(* IEC 61131-3 sources: SIMERLIFT/LOGICAD/SIMERLIFT/src_FBD/BCU/CAN/BCU, 3 files *)

(* ---- BCU_Battery_Status.iecfbd ---- *)
FUNCTION_BLOCK BCU_Battery_Status
  {
    SoC {index := 2};
    SoH {index := 3};
    Duty_Cycle {index := 4};
    Remain_Energy {index := 6};
    CAN_CH {index := 0};
    CAN_ID {index := 1};
    CAN_Error {index := 6};
    Available_Energy {index := 5};
    width := 500;
    height := 138;
    bgColor := "cadetblue";
  }

  VAR
    CANSEND4 : CANSEND;
  END_VAR
  VAR_INPUT
    SoC : USINT := 0;
    SoH : USINT := 0;
    Duty_Cycle : UINT := 0;
    Remain_Energy : REAL := 0;
    CAN_ID : UDINT := 0;
    CAN_CH : UDINT := 0;
    Available_Energy : REAL;
  END_VAR
  VAR_OUTPUT
    CAN_Error : BOOL := 0;
  END_VAR

  (*

    // Network 1:
    TO_LWORD(IN := SoC, TO_LWORD => @C(24).TO_LWORD);
    WBIT(start := 0, len := 8, INbit := @C(24).TO_LWORD, OUTbit => @C(2).OUTbit);
    TO_LWORD(IN := SoH, TO_LWORD => @C(31).TO_LWORD);
    WBIT(start := 8, len := 8, INbit := @C(31).TO_LWORD, OUTbit => @C(6).OUTbit);
    NE(IN1 := CAN_ID, IN2 := 0, NE => @C(64).NE);
    TO_LWORD(IN := Duty_Cycle, TO_LWORD => @C(32).TO_LWORD);
    WBIT(start := 16, len := 16, INbit := @C(32).TO_LWORD, OUTbit => @C(10).OUTbit);
    WFLT(start := 32, len := 16, prm := Remain_Energy, ofs := 0, res := 0.01, OUTbit => @C(14).OUTbit);
    WFLT(start := 48, len := 16, prm := Available_Energy, ofs := 0, res := 0.01, OUTbit => @C(15).OUTbit);
    OR(IN1 := @C(2).OUTbit, IN2 := @C(6).OUTbit, IN3 := @C(10).OUTbit, IN4 := @C(14).OUTbit, IN5 := @C(15).OUTbit, OR => @C(12).OR);
    CANSEND4(CH := CAN_CH, ID := CAN_ID, FMT := CAN_FORMAT#EXTENDED, DATA := @C(12).OR, DLC := 8, PER := T#100ms, ENB := @C(64).NE);
    NE(IN1 := CANSEND4.RC, IN2 := 0, NE => CAN_Error);

  *)

  @C(12) : @F(OR), @R(970.0, 60.0, 40.0, 108.0), LWORD, @I(@N(IN1), @L(9.5)), @I(@N(IN2), @L(29.5)), @I(@N(IN3), @L(49.5)), @I(@N(IN4), @L(69.5)), @I(@N(IN5), @L(89.5)), @O(@N(OR), @R(9.5));
  @VF(18) : @E(T#100ms), @R(1160.0, 160.0, 110.0, 19.0);
  @VF(19) : @E(8), @R(1160.0, 140.0, 110.0, 19.0), UDINT;
  @VF(20) : @E(CAN_FORMAT#EXTENDED), @R(1050.0, 120.0, 220.0, 19.0);
  @VF(25) : @E(16), @R(620.0, 200.0, 110.0, 19.0), INT;
  @VF(26) : @E(16), @R(620.0, 180.0, 110.0, 19.0), INT;
  @VF(27) : @E(8), @R(620.0, 140.0, 110.0, 19.0), INT;
  @VF(28) : @E(8), @R(620.0, 120.0, 110.0, 19.0), INT;
  @VF(29) : @E(8), @R(620.0, 80.0, 110.0, 19.0), INT;
  @VF(30) : @E(0), @R(620.0, 60.0, 110.0, 19.0), INT;
  @VF(35) : @E(16), @R(620.0, 260.0, 110.0, 19.0), INT;
  @VF(42) : @E(32), @R(620.0, 240.0, 110.0, 19.0), INT;
  @VF(3) : @E(SoC), @R(470.0, 100.0, 110.0, 19.0);
  @VF(4) : @E(SoH), @R(470.0, 160.0, 110.0, 19.0);
  @VF(5) : @E(Duty_Cycle), @R(470.0, 220.0, 110.0, 19.0);
  @VF(8) : @E(Remain_Energy), @R(470.0, 280.0, 150.0, 19.0);
  @VF(58) : @E(CAN_ID), @R(1050.0, 100.0, 220.0, 19.0);
  @C(64) : @F(NE), @R(1350.0, 180.0, 40.0, 38.0), UDINT, @I(@N(IN1), @L(9.5)), @I(@N(IN2), @L(29.5)), @O(@N(NE), @R(9.5));
  @VF(66) : @E(0), @R(1160.0, 200.0, 110.0, 19.0), UDINT;
  @VF(61) : @E(CAN_CH), @R(1050.0, 80.0, 220.0, 19.0);
  @C(95) : @F(NE), @R(1590.0, 180.0, 40.0, 38.0), UINT, @I(@N(IN1), @L(9.5)), @I(@N(IN2), @L(29.5)), @O(@N(NE), @R(9.5));
  @VF(114) : @E(CAN_Error), @R(1660.0, 180.0, 110.0, 19.0);
  @VF(115) : @E(0), @R(1440.0, 200.0, 110.0, 19.0), UINT;
  @C(11) : @FB(CANSEND4), @R(1430.0, 60.0, 120.0, 138.0), @I(@N(CH), @L(29.5)), @I(@N(ID), @L(49.5)), @I(@N(FMT), @L(69.5)), @I(@N(DATA), @L(9.5)), @I(@N(DLC), @L(89.5)), @I(@N(PER), @L(109.5)), @I(@N(ENB), @L(129.5)), @O(@N(CTX), @R(9.5)), @O(@N(RC), @R(129.5));
  @VF(13) : @E(16), @R(620.0, 360.0, 110.0, 19.0), INT;
  @VF(17) : @E(48), @R(620.0, 340.0, 110.0, 19.0), INT;
  @VF(71) : @E(Available_Energy), @R(470.0, 380.0, 150.0, 19.0);
  @C(2) : @F(WBIT), @R(790.0, 60.0, 120.0, 58.0), @I(@N(start), @L(9.5)), @I(@N(len), @L(29.5)), @I(@N(INbit), @L(49.5)), @O(@N(OUTbit), @R(9.5));
  @C(6) : @F(WBIT), @R(790.0, 120.0, 120.0, 58.0), @I(@N(start), @L(9.5)), @I(@N(len), @L(29.5)), @I(@N(INbit), @L(49.5)), @O(@N(OUTbit), @R(9.5));
  @C(10) : @F(WBIT), @R(790.0, 180.0, 120.0, 58.0), @I(@N(start), @L(9.5)), @I(@N(len), @L(29.5)), @I(@N(INbit), @L(49.5)), @O(@N(OUTbit), @R(9.5));
  @C(24) : @F(TO_LWORD), @R(610.0, 100.0, 120.0, 18.0), USINT, @I(@N(IN), @L(9.5)), @O(@N(TO_LWORD), @R(9.5));
  @C(31) : @F(TO_LWORD), @R(610.0, 160.0, 120.0, 18.0), USINT, @I(@N(IN), @L(9.5)), @O(@N(TO_LWORD), @R(9.5));
  @C(32) : @F(TO_LWORD), @R(610.0, 220.0, 120.0, 18.0), UINT, @I(@N(IN), @L(9.5)), @O(@N(TO_LWORD), @R(9.5));
  @C(14) : @F(WFLT), @R(790.0, 240.0, 120.0, 98.0), @I(@N(start), @L(9.5)), @I(@N(len), @L(29.5)), @I(@N(prm), @L(49.5)), @I(@N(ofs), @L(69.5)), @I(@N(res), @L(89.5)), @O(@N(OUTbit), @R(9.5));
  @C(15) : @F(WFLT), @R(790.0, 340.0, 120.0, 98.0), @I(@N(start), @L(9.5)), @I(@N(len), @L(29.5)), @I(@N(prm), @L(49.5)), @I(@N(ofs), @L(69.5)), @I(@N(res), @L(89.5)), @O(@N(OUTbit), @R(9.5));
  @VF(23) : @E(0), @R(680.0, 400.0, 50.0, 19.0), LREAL;
  @VF(41) : @E(0.01), @R(680.0, 420.0, 50.0, 19.0), LREAL;
  @VF(44) : @E(0.01), @R(680.0, 320.0, 50.0, 19.0), LREAL;
  @VF(45) : @E(0), @R(680.0, 300.0, 50.0, 19.0), LREAL;
  @CP(65) : 1309.5, 109.5;

  @G(34) :
     @L(@VF(18).o, @C(11).PER)
    ;
  @G(33) :
     @L(@VF(19).o, @C(11).DLC)
    ;
  @G(38) :
     @L(@VF(20).o, @C(11).FMT)
    ;
  @G(43) :
     @L(@C(12).OR, @C(11).DATA)
    ;
  @G(37) :
     @L(@VF(58).o, @CP(65)),
     @L(@CP(65), @C(11).ID),
     @L(@CP(65), @C(64).IN1)
    ;
  @G(67) :
     @L(@VF(66).o, @C(64).IN2)
    ;
  @G(1) :
     @L(@C(64).NE, @C(11).ENB)
    ;
  @G(7) :
     @L(@VF(61).o, @C(11).CH)
    ;
  @G(98) :
     @L(@VF(115).o, @C(95).IN2)
    ;
  @G(97) :
     @L(@C(95).NE, @VF(114).i)
    ;
  @G(9) :
     @L(@C(11).RC, @C(95).IN1)
    ;
  @G(57) :
     @L(@C(32).TO_LWORD, @C(10).INbit)
    ;
  @G(59) :
     @L(@VF(25).o, @C(10).len)
    ;
  @G(63) :
     @L(@VF(26).o, @C(10).start)
    ;
  @G(68) :
     @L(@C(31).TO_LWORD, @C(6).INbit)
    ;
  @G(69) :
     @L(@VF(27).o, @C(6).len)
    ;
  @G(70) :
     @L(@VF(28).o, @C(6).start)
    ;
  @G(72) :
     @L(@C(24).TO_LWORD, @C(2).INbit)
    ;
  @G(73) :
     @L(@VF(29).o, @C(2).len)
    ;
  @G(74) :
     @L(@VF(30).o, @C(2).start)
    ;
  @G(75) :
     @L(@C(2).OUTbit, @C(12).IN1)
    ;
  @G(76) :
     @L(@C(6).OUTbit, @C(12).IN2)
    ;
  @G(77) :
     @L(@C(10).OUTbit, @C(12).IN3)
    ;
  @G(82) :
     @L(@VF(3).o, @C(24).IN)
    ;
  @G(83) :
     @L(@VF(4).o, @C(31).IN)
    ;
  @G(84) :
     @L(@VF(5).o, @C(32).IN)
    ;
  @G(21) :
     @L(@VF(17).o, @C(15).start)
    ;
  @G(22) :
     @L(@VF(13).o, @C(15).len)
    ;
  @G(40) :
     @L(@VF(23).o, @C(15).ofs)
    ;
  @G(46) :
     @L(@VF(45).o, @C(14).ofs)
    ;
  @G(47) :
     @L(@VF(44).o, @C(14).res)
    ;
  @G(48) :
     @L(@VF(35).o, @C(14).len)
    ;
  @G(49) :
     @L(@VF(42).o, @C(14).start)
    ;
  @G(50) :
     @L(@VF(41).o, @C(15).res)
    ;
  @G(39) :
     @L(@C(14).OUTbit, @C(12).IN4)
    ;
  @G(51) :
     @L(@C(15).OUTbit, @C(12).IN5)
    ;
  @G(16) :
     @L(@VF(8).o, @C(14).prm)
    ;
  @G(36) :
     @L(@VF(71).o, @C(15).prm)
    ;
END_FUNCTION_BLOCK

(* ---- BCU_Cell_Status.iecfbd ---- *)
FUNCTION_BLOCK BCU_Cell_Status
  {
    Cell_Temp {loc := "left", index := 7};
    Cell_Voltage {loc := "left", index := 6};
    Selected_Cell_Loc {loc := "left", index := 5};
    Selected_BMU_Loc {loc := "left", index := 4};
    CAN_CH {index := 0};
    CAN_ID {index := 1};
    CAN_Error {index := 7};
    Total_Voltage {index := 2};
    Instant_Current {index := 3};
    width := 500;
    height := 158;
    bgColor := "cadetblue";
  }

  VAR
    CANSEND3 : CANSEND;
  END_VAR
  VAR_INPUT
    Selected_BMU_Loc : USINT := 0;
    Selected_Cell_Loc : USINT := 0;
    Cell_Voltage : UDINT := 0;
    Cell_Temp : REAL := 0;
    CAN_ID : UDINT := 0;
    CAN_CH : UDINT := 0;
    Total_Voltage : REAL := 0;
    Instant_Current : REAL := 0;
  END_VAR
  VAR_OUTPUT
    CAN_Error : BOOL := 0;
  END_VAR

  (*

    // Network 1:
    WFLT(start := 0, len := 16, prm := Total_Voltage, ofs := 0, res := 0.1, OUTbit => @C(7).OUTbit);
    WFLT(start := 16, len := 16, prm := Instant_Current, ofs := -1000, res := 0.1, OUTbit => @C(14).OUTbit);
    NE(IN1 := CAN_ID, IN2 := 0, NE => @C(64).NE);
    TO_LWORD(IN := Selected_BMU_Loc, TO_LWORD => @C(44).TO_LWORD);
    WBIT(start := 32, len := 4, INbit := @C(44).TO_LWORD, OUTbit => @C(15).OUTbit);
    TO_LWORD(IN := Selected_Cell_Loc, TO_LWORD => @C(47).TO_LWORD);
    WBIT(start := 36, len := 4, INbit := @C(47).TO_LWORD, OUTbit => @C(16).OUTbit);
    TO_LWORD(IN := Cell_Voltage, TO_LWORD => @C(48).TO_LWORD);
    WBIT(start := 40, len := 16, INbit := @C(48).TO_LWORD, OUTbit => @C(17).OUTbit);
    WFLT(start := 56, len := 8, prm := Cell_Temp, ofs := -40, res := 1, OUTbit => @C(20).OUTbit);
    OR(IN1 := @C(7).OUTbit, IN2 := @C(14).OUTbit, IN3 := @C(15).OUTbit, IN4 := @C(16).OUTbit, IN5 := @C(17).OUTbit, IN6 := @C(20).OUTbit, OR => @C(226).OR);
    CANSEND3(CH := CAN_CH, ID := CAN_ID, FMT := CAN_FORMAT#EXTENDED, DATA := @C(226).OR, DLC := 8, PER := T#100ms, ENB := @C(64).NE);
    NE(IN1 := CANSEND3.RC, IN2 := 0, NE => CAN_Error);

  *)

  @C(226) : @F(OR), @R(730.0, 40.0, 40.0, 118.0), LWORD, @I(@N(IN1), @L(9.5)), @I(@N(IN2), @L(29.5)), @I(@N(IN3), @L(49.5)), @I(@N(IN4), @L(69.5)), @I(@N(IN5), @L(89.5)), @I(@N(IN6), @L(109.5)), @O(@N(OR), @R(9.5));
  @VF(259) : @E(8), @R(920.0, 120.0, 110.0, 19.0), UDINT;
  @VF(258) : @E(T#100ms), @R(920.0, 140.0, 110.0, 19.0);
  @VF(262) : @E(CAN_FORMAT#EXTENDED), @R(810.0, 100.0, 220.0, 19.0);
  @VF(230) : @E(32), @R(380.0, 240.0, 110.0, 19.0), INT;
  @VF(231) : @E(4), @R(380.0, 260.0, 110.0, 19.0), INT;
  @VF(232) : @E(36), @R(380.0, 300.0, 110.0, 19.0), INT;
  @VF(233) : @E(4), @R(380.0, 320.0, 110.0, 19.0), INT;
  @VF(234) : @E(40), @R(380.0, 360.0, 110.0, 19.0), INT;
  @VF(235) : @E(16), @R(380.0, 380.0, 110.0, 19.0), INT;
  @VF(236) : @E(56), @R(380.0, 420.0, 110.0, 19.0), INT;
  @VF(237) : @E(8), @R(380.0, 440.0, 110.0, 19.0), INT;
  @VF(228) : @E(-40), @R(380.0, 480.0, 110.0, 19.0), LREAL;
  @VF(250) : @E(1), @R(380.0, 500.0, 110.0, 19.0), LREAL;
  @VF(3) : @E(Selected_BMU_Loc), @R(40.0, 280.0, 220.0, 19.0);
  @VF(4) : @E(Selected_Cell_Loc), @R(40.0, 340.0, 220.0, 19.0);
  @VF(5) : @E(Cell_Voltage), @R(40.0, 400.0, 220.0, 19.0);
  @VF(6) : @E(Cell_Temp), @R(40.0, 460.0, 220.0, 19.0);
  @VF(1) : @E(CAN_ID), @R(810.0, 80.0, 220.0, 19.0);
  @C(64) : @F(NE), @R(1110.0, 160.0, 40.0, 38.0), UDINT, @I(@N(IN1), @L(9.5)), @I(@N(IN2), @L(29.5)), @O(@N(NE), @R(9.5));
  @VF(66) : @E(0), @R(920.0, 180.0, 110.0, 19.0), UDINT;
  @VF(18) : @E(CAN_CH), @R(810.0, 60.0, 220.0, 19.0);
  @C(95) : @F(NE), @R(1330.0, 160.0, 40.0, 38.0), UINT, @I(@N(IN1), @L(9.5)), @I(@N(IN2), @L(29.5)), @O(@N(NE), @R(9.5));
  @VF(114) : @E(CAN_Error), @R(1390.0, 160.0, 110.0, 19.0);
  @VF(115) : @E(0), @R(1200.0, 180.0, 110.0, 19.0), UINT;
  @VF(36) : @E(16), @R(380.0, 160.0, 110.0, 19.0), INT;
  @VF(37) : @E(16), @R(380.0, 140.0, 110.0, 19.0), INT;
  @VF(38) : @E(16), @R(380.0, 60.0, 110.0, 19.0), INT;
  @VF(39) : @E(0), @R(380.0, 40.0, 110.0, 19.0), INT;
  @VF(166) : @E(0.1), @R(380.0, 220.0, 110.0, 19.0), LREAL;
  @VF(165) : @E(-1000), @R(380.0, 200.0, 110.0, 19.0), LREAL;
  @VF(40) : @E(Total_Voltage), @R(40.0, 80.0, 220.0, 19.0);
  @VF(41) : @E(Instant_Current), @R(40.0, 180.0, 220.0, 19.0);
  @VF(45) : @E(0), @R(380.0, 100.0, 110.0, 19.0), LREAL;
  @VF(46) : @E(0.1), @R(380.0, 120.0, 110.0, 19.0), LREAL;
  @C(158) : @FB(CANSEND3), @R(1190.0, 40.0, 120.0, 138.0), @I(@N(CH), @L(29.5)), @I(@N(ID), @L(49.5)), @I(@N(FMT), @L(69.5)), @I(@N(DATA), @L(9.5)), @I(@N(DLC), @L(89.5)), @I(@N(PER), @L(109.5)), @I(@N(ENB), @L(129.5)), @O(@N(CTX), @R(9.5)), @O(@N(RC), @R(129.5));
  @C(7) : @F(WFLT), @R(540.0, 40.0, 120.0, 98.0), @I(@N(start), @L(9.5)), @I(@N(len), @L(29.5)), @I(@N(prm), @L(49.5)), @I(@N(ofs), @L(69.5)), @I(@N(res), @L(89.5)), @O(@N(OUTbit), @R(9.5));
  @C(14) : @F(WFLT), @R(540.0, 140.0, 120.0, 98.0), @I(@N(start), @L(9.5)), @I(@N(len), @L(29.5)), @I(@N(prm), @L(49.5)), @I(@N(ofs), @L(69.5)), @I(@N(res), @L(89.5)), @O(@N(OUTbit), @R(9.5));
  @C(15) : @F(WBIT), @R(540.0, 240.0, 120.0, 58.0), @I(@N(start), @L(9.5)), @I(@N(len), @L(29.5)), @I(@N(INbit), @L(49.5)), @O(@N(OUTbit), @R(9.5));
  @C(16) : @F(WBIT), @R(540.0, 300.0, 120.0, 58.0), @I(@N(start), @L(9.5)), @I(@N(len), @L(29.5)), @I(@N(INbit), @L(49.5)), @O(@N(OUTbit), @R(9.5));
  @C(17) : @F(WBIT), @R(540.0, 360.0, 120.0, 58.0), @I(@N(start), @L(9.5)), @I(@N(len), @L(29.5)), @I(@N(INbit), @L(49.5)), @O(@N(OUTbit), @R(9.5));
  @C(20) : @F(WFLT), @R(540.0, 420.0, 120.0, 98.0), @I(@N(start), @L(9.5)), @I(@N(len), @L(29.5)), @I(@N(prm), @L(49.5)), @I(@N(ofs), @L(69.5)), @I(@N(res), @L(89.5)), @O(@N(OUTbit), @R(9.5));
  @C(44) : @F(TO_LWORD), @R(370.0, 280.0, 120.0, 18.0), USINT, @I(@N(IN), @L(9.5)), @O(@N(TO_LWORD), @R(9.5));
  @C(47) : @F(TO_LWORD), @R(370.0, 340.0, 120.0, 18.0), USINT, @I(@N(IN), @L(9.5)), @O(@N(TO_LWORD), @R(9.5));
  @C(48) : @F(TO_LWORD), @R(370.0, 400.0, 120.0, 18.0), UDINT, @I(@N(IN), @L(9.5)), @O(@N(TO_LWORD), @R(9.5));
  @CP(12) : 1069.5, 89.5;

  @G(239) :
     @L(@VF(262).o, @C(158).FMT)
    ;
  @G(253) :
     @L(@VF(259).o, @C(158).DLC)
    ;
  @G(254) :
     @L(@VF(258).o, @C(158).PER)
    ;
  @G(161) :
     @L(@C(226).OR, @C(158).DATA)
    ;
  @G(2) :
     @L(@VF(1).o, @CP(12)),
     @L(@CP(12), @C(158).ID),
     @L(@CP(12), @C(64).IN1)
    ;
  @G(67) :
     @L(@VF(66).o, @C(64).IN2)
    ;
  @G(11) :
     @L(@C(64).NE, @C(158).ENB)
    ;
  @G(13) :
     @L(@VF(18).o, @C(158).CH)
    ;
  @G(98) :
     @L(@VF(115).o, @C(95).IN2)
    ;
  @G(97) :
     @L(@C(95).NE, @VF(114).i)
    ;
  @G(19) :
     @L(@C(158).RC, @C(95).IN1)
    ;
  @G(9) :
     @L(@VF(45).o, @C(7).ofs)
    ;
  @G(10) :
     @L(@VF(46).o, @C(7).res)
    ;
  @G(23) :
     @L(@VF(39).o, @C(7).start)
    ;
  @G(30) :
     @L(@VF(38).o, @C(7).len)
    ;
  @G(31) :
     @L(@VF(37).o, @C(14).start)
    ;
  @G(32) :
     @L(@VF(36).o, @C(14).len)
    ;
  @G(34) :
     @L(@VF(165).o, @C(14).ofs)
    ;
  @G(35) :
     @L(@VF(166).o, @C(14).res)
    ;
  @G(42) :
     @L(@VF(230).o, @C(15).start)
    ;
  @G(43) :
     @L(@VF(231).o, @C(15).len)
    ;
  @G(49) :
     @L(@C(44).TO_LWORD, @C(15).INbit)
    ;
  @G(50) :
     @L(@VF(232).o, @C(16).start)
    ;
  @G(51) :
     @L(@VF(233).o, @C(16).len)
    ;
  @G(52) :
     @L(@C(47).TO_LWORD, @C(16).INbit)
    ;
  @G(53) :
     @L(@VF(234).o, @C(17).start)
    ;
  @G(54) :
     @L(@VF(235).o, @C(17).len)
    ;
  @G(55) :
     @L(@C(48).TO_LWORD, @C(17).INbit)
    ;
  @G(56) :
     @L(@VF(236).o, @C(20).start)
    ;
  @G(57) :
     @L(@VF(237).o, @C(20).len)
    ;
  @G(58) :
     @L(@VF(6).o, @C(20).prm)
    ;
  @G(59) :
     @L(@VF(228).o, @C(20).ofs)
    ;
  @G(60) :
     @L(@VF(250).o, @C(20).res)
    ;
  @G(61) :
     @L(@VF(5).o, @C(48).IN)
    ;
  @G(62) :
     @L(@VF(4).o, @C(47).IN)
    ;
  @G(63) :
     @L(@VF(3).o, @C(44).IN)
    ;
  @G(65) :
     @L(@C(7).OUTbit, @C(226).IN1)
    ;
  @G(68) :
     @L(@C(14).OUTbit, @C(226).IN2)
    ;
  @G(69) :
     @L(@C(15).OUTbit, @C(226).IN3)
    ;
  @G(70) :
     @L(@C(16).OUTbit, @C(226).IN4)
    ;
  @G(71) :
     @L(@C(17).OUTbit, @C(226).IN5)
    ;
  @G(72) :
     @L(@C(20).OUTbit, @C(226).IN6)
    ;
  @G(8) :
     @L(@VF(40).o, @C(7).prm)
    ;
  @G(21) :
     @L(@VF(41).o, @C(14).prm)
    ;
END_FUNCTION_BLOCK

(* ---- BCU_State_Message.iecfbd ---- *)
FUNCTION_BLOCK BCU_State_Message
  {
    DMDC {loc := "left", index := 6};
    Ambient_Temp {loc := "left", index := 5};
    ChargeContact {loc := "left", index := 4};
    Contactor_Status {loc := "left", index := 3};
    State {loc := "left", index := 2};
    DMCC {index := 7};
    CAN_CH {index := 0};
    CAN_ID {index := 1};
    CAN_Error {index := 7};
    width := 500;
    height := 158;
    bgColor := "cadetblue";
  }

  VAR
    CANSEND4 : CANSEND;
  END_VAR
  VAR_INPUT
    CAN_ID : UDINT := 0;
    State : USINT := 0;
    Contactor_Status : BOOL := 0;
    ChargeContact : BOOL := 0;
    Ambient_Temp : REAL := 0;
    DMDC : UINT := 0;
    DMCC : UINT := 0;
    CAN_CH : UDINT := 0;
    NegContact : BOOL;
    isolationStatus : USINT;
    chargeComplete : BOOL;
    dischargeComplete : BOOL;
    emergencyButton : BOOL;
    in1Status : USINT;
    in2Status : USINT;
  END_VAR
  VAR_OUTPUT
    CAN_Error : BOOL := 0;
  END_VAR

  (*

    // Network 1:
    TO_LWORD(IN := State, TO_LWORD => @C(16).TO_LWORD);
    WBIT(start := 0, len := 8, INbit := @C(16).TO_LWORD, OUTbit => @C(2).OUTbit);
    TO_LWORD(IN := Contactor_Status, TO_LWORD => @C(17).TO_LWORD);
    WBIT(start := 8, len := 1, INbit := @C(17).TO_LWORD, OUTbit => @C(9).OUTbit);
    NE(IN1 := CAN_ID, IN2 := 0, NE => @C(64).NE);
    TO_LWORD(IN := ChargeContact, TO_LWORD => @C(86).TO_LWORD);
    WBIT(start := 9, len := 1, INbit := @C(86).TO_LWORD, OUTbit => @C(87).OUTbit);
    TO_LWORD(IN := NegContact, TO_LWORD => @C(79).TO_LWORD);
    WBIT(start := 10, len := 1, INbit := @C(79).TO_LWORD, OUTbit => @C(81).OUTbit);
    TO_LWORD(IN := chargeComplete, TO_LWORD => @C(104).TO_LWORD);
    WBIT(start := 11, len := 1, INbit := @C(104).TO_LWORD, OUTbit => @C(105).OUTbit);
    TO_LWORD(IN := dischargeComplete, TO_LWORD => @C(120).TO_LWORD);
    WBIT(start := 12, len := 1, INbit := @C(120).TO_LWORD, OUTbit => @C(121).OUTbit);
    TO_LWORD(IN := emergencyButton, TO_LWORD => @C(129).TO_LWORD);
    WBIT(start := 13, len := 1, INbit := @C(129).TO_LWORD, OUTbit => @C(130).OUTbit);
    TO_LWORD(IN := isolationStatus, TO_LWORD => @C(13).TO_LWORD);
    WBIT(start := 14, len := 2, INbit := @C(13).TO_LWORD, OUTbit => @C(3).OUTbit);
    TO_LWORD(IN := in1Status, TO_LWORD => @C(138).TO_LWORD);
    WBIT(start := 16, len := 2, INbit := @C(138).TO_LWORD, OUTbit => @C(139).OUTbit);
    TO_LWORD(IN := in2Status, TO_LWORD => @C(147).TO_LWORD);
    WBIT(start := 18, len := 2, INbit := @C(147).TO_LWORD, OUTbit => @C(148).OUTbit);
    WFLT(start := 24, len := 8, prm := Ambient_Temp, ofs := -40, res := 1, OUTbit => @C(10).OUTbit);
    WFLT(start := 32, len := 16, prm := DMCC, ofs := 0, res := 0.1, OUTbit => @C(15).OUTbit);
    WFLT(start := 48, len := 12, prm := DMDC, ofs := 0, res := 0.1, OUTbit => @C(14).OUTbit);
    OR(IN1 := @C(2).OUTbit, IN2 := @C(9).OUTbit, IN3 := @C(87).OUTbit, IN4 := @C(81).OUTbit, IN5 := @C(105).OUTbit, IN6 := @C(121).OUTbit, IN7 := @C(130).OUTbit, IN8 := @C(3).OUTbit, IN9 := @C(139).OUTbit, IN10 := @C(148).OUTbit, IN11 := @C(10).OUTbit, IN12 := @C(15).OUTbit, IN13 := @C(14).OUTbit, OR => @C(12).OR);
    CANSEND4(CH := CAN_CH, ID := CAN_ID, FMT := CAN_FORMAT#EXTENDED, DATA := @C(12).OR, DLC := 8, PER := T#100ms, ENB := @C(64).NE);
    NE(IN1 := CANSEND4.RC, IN2 := 0, NE => CAN_Error);

  *)

  @C(64) : @F(NE), @R(1110.0, 170.0, 40.0, 38.0), UDINT, @I(@N(IN1), @L(9.5)), @I(@N(IN2), @L(29.5)), @O(@N(NE), @R(9.5));
  @C(12) : @F(OR), @R(760.0, 50.0, 40.0, 258.0), LWORD, @I(@N(IN1), @L(9.5)), @I(@N(IN2), @L(29.5)), @I(@N(IN3), @L(49.5)), @I(@N(IN4), @L(69.5)), @I(@N(IN5), @L(89.5)), @I(@N(IN6), @L(109.5)), @I(@N(IN7), @L(129.5)), @I(@N(IN8), @L(149.5)), @I(@N(IN9), @L(169.5)), @I(@N(IN10), @L(189.5)), @I(@N(IN11), @L(209.5)), @I(@N(IN12), @L(229.5)), @I(@N(IN13), @L(249.5)), @O(@N(OR), @R(9.5));
  @VF(66) : @E(0), @R(920.0, 190.0, 110.0, 19.0), UDINT;
  @VF(18) : @E(T#100ms), @R(920.0, 150.0, 110.0, 19.0);
  @VF(19) : @E(8), @R(920.0, 130.0, 110.0, 19.0), UDINT;
  @VF(20) : @E(CAN_FORMAT#EXTENDED), @R(810.0, 110.0, 220.0, 19.0);
  @VF(58) : @E(CAN_ID), @R(810.0, 90.0, 220.0, 19.0);
  @VF(25) : @E(1), @R(410.0, 130.0, 110.0, 19.0), INT;
  @VF(27) : @E(2), @R(410.0, 490.0, 110.0, 19.0), INT;
  @VF(26) : @E(8), @R(410.0, 110.0, 110.0, 19.0), INT;
  @VF(29) : @E(8), @R(410.0, 70.0, 110.0, 19.0), INT;
  @VF(28) : @E(14), @R(410.0, 470.0, 110.0, 19.0), INT;
  @VF(30) : @E(0), @R(410.0, 50.0, 110.0, 19.0), INT;
  @VF(35) : @E(8), @R(410.0, 670.0, 110.0, 19.0), INT;
  @VF(42) : @E(24), @R(410.0, 650.0, 110.0, 19.0), INT;
  @VF(55) : @E(48), @R(410.0, 850.0, 110.0, 19.0), INT;
  @VF(54) : @E(12), @R(410.0, 870.0, 110.0, 19.0), INT;
  @VF(4) : @E(State), @R(230.0, 90.0, 140.0, 19.0);
  @VF(5) : @E(Contactor_Status), @R(220.0, 150.0, 150.0, 19.0);
  @VF(6) : @E(ChargeContact), @R(230.0, 210.0, 140.0, 19.0);
  @VF(7) : @E(Ambient_Temp), @R(230.0, 690.0, 140.0, 19.0);
  @VF(8) : @E(DMDC), @R(230.0, 890.0, 140.0, 19.0);
  @VF(60) : @E(16), @R(410.0, 770.0, 110.0, 19.0), INT;
  @VF(61) : @E(32), @R(410.0, 750.0, 110.0, 19.0), INT;
  @VF(68) : @E(DMCC), @R(230.0, 790.0, 140.0, 19.0);
  @VF(71) : @E(CAN_CH), @R(810.0, 70.0, 220.0, 19.0);
  @VF(69) : @E(0), @R(410.0, 910.0, 110.0, 19.0), LREAL;
  @VF(70) : @E(0.1), @R(410.0, 930.0, 110.0, 19.0), LREAL;
  @VF(74) : @E(0), @R(410.0, 810.0, 110.0, 19.0), LREAL;
  @VF(75) : @E(0.1), @R(410.0, 830.0, 110.0, 19.0), LREAL;
  @C(95) : @F(NE), @R(1350.0, 170.0, 40.0, 38.0), UINT, @I(@N(IN1), @L(9.5)), @I(@N(IN2), @L(29.5)), @O(@N(NE), @R(9.5));
  @VF(114) : @E(CAN_Error), @R(1420.0, 170.0, 110.0, 19.0);
  @VF(115) : @E(0), @R(1200.0, 190.0, 110.0, 19.0), UINT;
  @VF(52) : @E(-40), @R(460.0, 710.0, 60.0, 19.0), LREAL;
  @VF(80) : @E(1), @R(460.0, 730.0, 60.0, 19.0), LREAL;
  @C(11) : @FB(CANSEND4), @R(1190.0, 50.0, 120.0, 138.0), @I(@N(CH), @L(29.5)), @I(@N(ID), @L(49.5)), @I(@N(FMT), @L(69.5)), @I(@N(DATA), @L(9.5)), @I(@N(DLC), @L(89.5)), @I(@N(PER), @L(109.5)), @I(@N(ENB), @L(129.5)), @O(@N(CTX), @R(9.5)), @O(@N(RC), @R(129.5));
  @C(2) : @F(WBIT), @R(560.0, 50.0, 120.0, 58.0), @I(@N(start), @L(9.5)), @I(@N(len), @L(29.5)), @I(@N(INbit), @L(49.5)), @O(@N(OUTbit), @R(9.5));
  @C(3) : @F(WBIT), @R(560.0, 470.0, 120.0, 58.0), @I(@N(start), @L(9.5)), @I(@N(len), @L(29.5)), @I(@N(INbit), @L(49.5)), @O(@N(OUTbit), @R(9.5));
  @C(9) : @F(WBIT), @R(560.0, 110.0, 120.0, 58.0), @I(@N(start), @L(9.5)), @I(@N(len), @L(29.5)), @I(@N(INbit), @L(49.5)), @O(@N(OUTbit), @R(9.5));
  @C(10) : @F(WFLT), @R(560.0, 650.0, 120.0, 98.0), @I(@N(start), @L(9.5)), @I(@N(len), @L(29.5)), @I(@N(prm), @L(49.5)), @I(@N(ofs), @L(69.5)), @I(@N(res), @L(89.5)), @O(@N(OUTbit), @R(9.5));
  @C(14) : @F(WFLT), @R(560.0, 850.0, 120.0, 98.0), @I(@N(start), @L(9.5)), @I(@N(len), @L(29.5)), @I(@N(prm), @L(49.5)), @I(@N(ofs), @L(69.5)), @I(@N(res), @L(89.5)), @O(@N(OUTbit), @R(9.5));
  @C(15) : @F(WFLT), @R(560.0, 750.0, 120.0, 98.0), @I(@N(start), @L(9.5)), @I(@N(len), @L(29.5)), @I(@N(prm), @L(49.5)), @I(@N(ofs), @L(69.5)), @I(@N(res), @L(89.5)), @O(@N(OUTbit), @R(9.5));
  @C(16) : @F(TO_LWORD), @R(400.0, 90.0, 120.0, 18.0), USINT, @I(@N(IN), @L(9.5)), @O(@N(TO_LWORD), @R(9.5));
  @C(13) : @F(TO_LWORD), @R(400.0, 510.0, 120.0, 18.0), USINT, @I(@N(IN), @L(9.5)), @O(@N(TO_LWORD), @R(9.5));
  @C(17) : @F(TO_LWORD), @R(400.0, 150.0, 120.0, 18.0), BOOL, @I(@N(IN), @L(9.5)), @O(@N(TO_LWORD), @R(9.5));
  @C(86) : @F(TO_LWORD), @R(400.0, 210.0, 120.0, 18.0), BOOL, @I(@N(IN), @L(9.5)), @O(@N(TO_LWORD), @R(9.5));
  @C(87) : @F(WBIT), @R(560.0, 170.0, 120.0, 58.0), @I(@N(start), @L(9.5)), @I(@N(len), @L(29.5)), @I(@N(INbit), @L(49.5)), @O(@N(OUTbit), @R(9.5));
  @VF(88) : @E(1), @R(410.0, 190.0, 110.0, 19.0), INT;
  @VF(89) : @E(9), @R(410.0, 170.0, 110.0, 19.0), INT;
  @VF(90) : @E(NegContact), @R(230.0, 270.0, 140.0, 19.0);
  @C(79) : @F(TO_LWORD), @R(400.0, 270.0, 120.0, 18.0), BOOL, @I(@N(IN), @L(9.5)), @O(@N(TO_LWORD), @R(9.5));
  @C(81) : @F(WBIT), @R(560.0, 230.0, 120.0, 58.0), @I(@N(start), @L(9.5)), @I(@N(len), @L(29.5)), @I(@N(INbit), @L(49.5)), @O(@N(OUTbit), @R(9.5));
  @VF(82) : @E(1), @R(410.0, 250.0, 110.0, 19.0), INT;
  @VF(107) : @E(isolationStatus), @R(230.0, 510.0, 140.0, 19.0);
  @VF(108) : @E(10), @R(410.0, 230.0, 110.0, 19.0), INT;
  @C(104) : @F(TO_LWORD), @R(400.0, 330.0, 120.0, 18.0), BOOL, @I(@N(IN), @L(9.5)), @O(@N(TO_LWORD), @R(9.5));
  @C(105) : @F(WBIT), @R(560.0, 290.0, 120.0, 58.0), @I(@N(start), @L(9.5)), @I(@N(len), @L(29.5)), @I(@N(INbit), @L(49.5)), @O(@N(OUTbit), @R(9.5));
  @VF(106) : @E(1), @R(410.0, 310.0, 110.0, 19.0), INT;
  @VF(112) : @E(11), @R(410.0, 290.0, 110.0, 19.0), INT;
  @VF(113) : @E(chargeComplete), @R(230.0, 330.0, 140.0, 19.0);
  @C(120) : @F(TO_LWORD), @R(400.0, 390.0, 120.0, 18.0), BOOL, @I(@N(IN), @L(9.5)), @O(@N(TO_LWORD), @R(9.5));
  @C(121) : @F(WBIT), @R(560.0, 350.0, 120.0, 58.0), @I(@N(start), @L(9.5)), @I(@N(len), @L(29.5)), @I(@N(INbit), @L(49.5)), @O(@N(OUTbit), @R(9.5));
  @VF(122) : @E(1), @R(410.0, 370.0, 110.0, 19.0), INT;
  @VF(123) : @E(12), @R(410.0, 350.0, 110.0, 19.0), INT;
  @VF(124) : @E(dischargeComplete), @R(230.0, 390.0, 140.0, 19.0);
  @C(129) : @F(TO_LWORD), @R(400.0, 450.0, 120.0, 18.0), BOOL, @I(@N(IN), @L(9.5)), @O(@N(TO_LWORD), @R(9.5));
  @C(130) : @F(WBIT), @R(560.0, 410.0, 120.0, 58.0), @I(@N(start), @L(9.5)), @I(@N(len), @L(29.5)), @I(@N(INbit), @L(49.5)), @O(@N(OUTbit), @R(9.5));
  @VF(131) : @E(1), @R(410.0, 430.0, 110.0, 19.0), INT;
  @VF(132) : @E(13), @R(410.0, 410.0, 110.0, 19.0), INT;
  @VF(133) : @E(emergencyButton), @R(230.0, 450.0, 140.0, 19.0);
  @C(138) : @F(TO_LWORD), @R(400.0, 570.0, 120.0, 18.0), USINT, @I(@N(IN), @L(9.5)), @O(@N(TO_LWORD), @R(9.5));
  @C(139) : @F(WBIT), @R(560.0, 530.0, 120.0, 58.0), @I(@N(start), @L(9.5)), @I(@N(len), @L(29.5)), @I(@N(INbit), @L(49.5)), @O(@N(OUTbit), @R(9.5));
  @VF(140) : @E(2), @R(410.0, 550.0, 110.0, 19.0), INT;
  @VF(141) : @E(16), @R(410.0, 530.0, 110.0, 19.0), INT;
  @VF(142) : @E(in1Status), @R(230.0, 570.0, 140.0, 19.0);
  @C(147) : @F(TO_LWORD), @R(400.0, 630.0, 120.0, 18.0), USINT, @I(@N(IN), @L(9.5)), @O(@N(TO_LWORD), @R(9.5));
  @C(148) : @F(WBIT), @R(560.0, 590.0, 120.0, 58.0), @I(@N(start), @L(9.5)), @I(@N(len), @L(29.5)), @I(@N(INbit), @L(49.5)), @O(@N(OUTbit), @R(9.5));
  @VF(149) : @E(2), @R(410.0, 610.0, 110.0, 19.0), INT;
  @VF(150) : @E(18), @R(410.0, 590.0, 110.0, 19.0), INT;
  @VF(151) : @E(in2Status), @R(230.0, 630.0, 140.0, 19.0);
  @CP(65) : 1069.5, 99.5;

  @G(67) :
     @L(@VF(66).o, @C(64).IN2)
    ;
  @G(1) :
     @L(@C(64).NE, @C(11).ENB)
    ;
  @G(34) :
     @L(@VF(18).o, @C(11).PER)
    ;
  @G(33) :
     @L(@VF(19).o, @C(11).DLC)
    ;
  @G(38) :
     @L(@VF(20).o, @C(11).FMT)
    ;
  @G(37) :
     @L(@VF(58).o, @CP(65)),
     @L(@CP(65), @C(11).ID),
     @L(@CP(65), @C(64).IN1)
    ;
  @G(43) :
     @L(@C(12).OR, @C(11).DATA)
    ;
  @G(22) :
     @L(@VF(71).o, @C(11).CH)
    ;
  @G(97) :
     @L(@C(95).NE, @VF(114).i)
    ;
  @G(98) :
     @L(@VF(115).o, @C(95).IN2)
    ;
  @G(78) :
     @L(@C(11).RC, @C(95).IN1)
    ;
  @G(21) :
     @L(@VF(30).o, @C(2).start)
    ;
  @G(23) :
     @L(@VF(29).o, @C(2).len)
    ;
  @G(24) :
     @L(@C(16).TO_LWORD, @C(2).INbit)
    ;
  @G(31) :
     @L(@VF(28).o, @C(3).start)
    ;
  @G(32) :
     @L(@VF(27).o, @C(3).len)
    ;
  @G(36) :
     @L(@C(13).TO_LWORD, @C(3).INbit)
    ;
  @G(39) :
     @L(@VF(26).o, @C(9).start)
    ;
  @G(40) :
     @L(@VF(25).o, @C(9).len)
    ;
  @G(41) :
     @L(@C(17).TO_LWORD, @C(9).INbit)
    ;
  @G(44) :
     @L(@VF(42).o, @C(10).start)
    ;
  @G(45) :
     @L(@VF(35).o, @C(10).len)
    ;
  @G(46) :
     @L(@VF(7).o, @C(10).prm)
    ;
  @G(47) :
     @L(@VF(52).o, @C(10).ofs)
    ;
  @G(48) :
     @L(@VF(80).o, @C(10).res)
    ;
  @G(49) :
     @L(@VF(55).o, @C(14).start)
    ;
  @G(50) :
     @L(@VF(54).o, @C(14).len)
    ;
  @G(51) :
     @L(@VF(8).o, @C(14).prm)
    ;
  @G(53) :
     @L(@VF(69).o, @C(14).ofs)
    ;
  @G(56) :
     @L(@VF(70).o, @C(14).res)
    ;
  @G(57) :
     @L(@VF(61).o, @C(15).start)
    ;
  @G(59) :
     @L(@VF(60).o, @C(15).len)
    ;
  @G(62) :
     @L(@VF(68).o, @C(15).prm)
    ;
  @G(63) :
     @L(@VF(74).o, @C(15).ofs)
    ;
  @G(72) :
     @L(@VF(75).o, @C(15).res)
    ;
  @G(73) :
     @L(@C(2).OUTbit, @C(12).IN1)
    ;
  @G(83) :
     @L(@VF(4).o, @C(16).IN)
    ;
  @G(91) :
     @L(@C(86).TO_LWORD, @C(87).INbit)
    ;
  @G(92) :
     @L(@VF(88).o, @C(87).len)
    ;
  @G(94) :
     @L(@VF(89).o, @C(87).start)
    ;
  @G(109) :
     @L(@C(79).TO_LWORD, @C(81).INbit)
    ;
  @G(110) :
     @L(@VF(82).o, @C(81).len)
    ;
  @G(111) :
     @L(@VF(108).o, @C(81).start)
    ;
  @G(85) :
     @L(@VF(90).o, @C(79).IN)
    ;
  @G(93) :
     @L(@VF(6).o, @C(86).IN)
    ;
  @G(103) :
     @L(@VF(5).o, @C(17).IN)
    ;
  @G(116) :
     @L(@C(104).TO_LWORD, @C(105).INbit)
    ;
  @G(117) :
     @L(@VF(106).o, @C(105).len)
    ;
  @G(118) :
     @L(@VF(112).o, @C(105).start)
    ;
  @G(119) :
     @L(@VF(113).o, @C(104).IN)
    ;
  @G(125) :
     @L(@C(120).TO_LWORD, @C(121).INbit)
    ;
  @G(126) :
     @L(@VF(122).o, @C(121).len)
    ;
  @G(127) :
     @L(@VF(123).o, @C(121).start)
    ;
  @G(128) :
     @L(@VF(124).o, @C(120).IN)
    ;
  @G(134) :
     @L(@C(129).TO_LWORD, @C(130).INbit)
    ;
  @G(135) :
     @L(@VF(131).o, @C(130).len)
    ;
  @G(136) :
     @L(@VF(132).o, @C(130).start)
    ;
  @G(137) :
     @L(@VF(133).o, @C(129).IN)
    ;
  @G(143) :
     @L(@C(138).TO_LWORD, @C(139).INbit)
    ;
  @G(144) :
     @L(@VF(140).o, @C(139).len)
    ;
  @G(145) :
     @L(@VF(141).o, @C(139).start)
    ;
  @G(146) :
     @L(@VF(142).o, @C(138).IN)
    ;
  @G(152) :
     @L(@C(147).TO_LWORD, @C(148).INbit)
    ;
  @G(153) :
     @L(@VF(149).o, @C(148).len)
    ;
  @G(154) :
     @L(@VF(150).o, @C(148).start)
    ;
  @G(155) :
     @L(@VF(151).o, @C(147).IN)
    ;
  @G(76) :
     @L(@VF(107).o, @C(13).IN)
    ;
  @G(77) :
     @L(@C(9).OUTbit, @C(12).IN2)
    ;
  @G(84) :
     @L(@C(87).OUTbit, @C(12).IN3)
    ;
  @G(96) :
     @L(@C(81).OUTbit, @C(12).IN4)
    ;
  @G(99) :
     @L(@C(105).OUTbit, @C(12).IN5)
    ;
  @G(100) :
     @L(@C(121).OUTbit, @C(12).IN6)
    ;
  @G(101) :
     @L(@C(130).OUTbit, @C(12).IN7)
    ;
  @G(102) :
     @L(@C(3).OUTbit, @C(12).IN8)
    ;
  @G(156) :
     @L(@C(139).OUTbit, @C(12).IN9)
    ;
  @G(157) :
     @L(@C(148).OUTbit, @C(12).IN10)
    ;
  @G(158) :
     @L(@C(10).OUTbit, @C(12).IN11)
    ;
  @G(159) :
     @L(@C(15).OUTbit, @C(12).IN12)
    ;
  @G(160) :
     @L(@C(14).OUTbit, @C(12).IN13)
    ;
END_FUNCTION_BLOCK
